RoboDK station: Pick&Place_UR5e.rdk

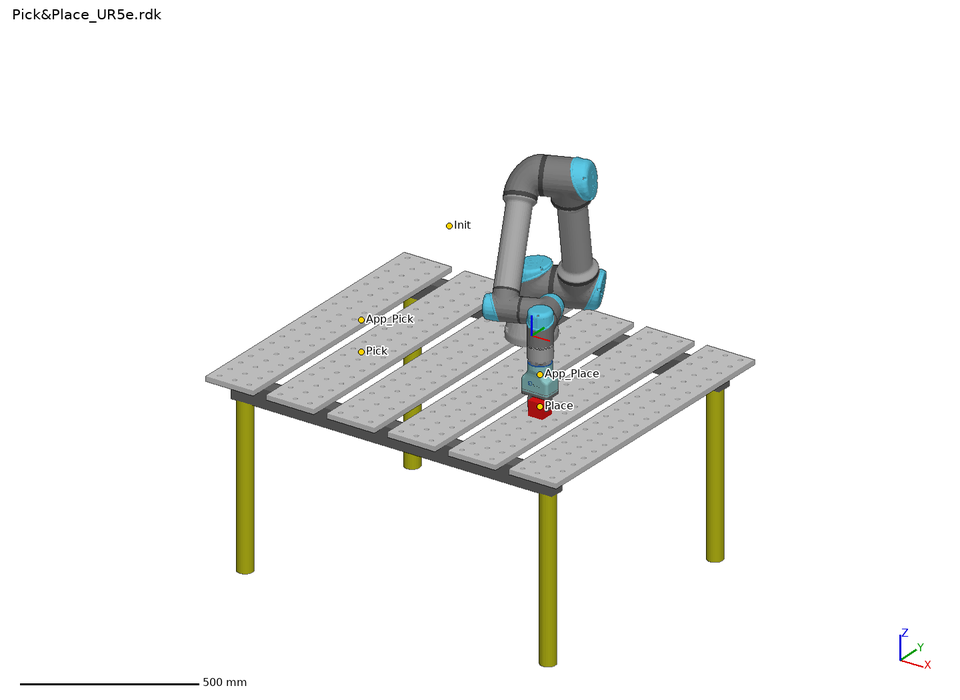
[picture v0: the station drawn from its stored meshes, robots at their saved joint values, targets as dots, program paths as lines]
Station Pick&Place_UR5e (saved by RoboDK 5.9.2). Poses are relative to the parent item; angles as X-Y-Z fixed-axis rotations.
  - frame UR5e Base at (0, 0, 0) mm
    - robot UR5e: 6 axes, payload 5 kg, reach 850 mm, repeatability 0.03 mm, weight 18.4 kg
        modified DH rows (alpha deg, a mm, theta deg, d mm): 0, 0, 0, 162.5; 90, 0, 180, 0; 0, 425, 0, 0; 0, 392.25, 0, 133.3; -90, 0, 0, 99.7; 90, 0, 180, 99.6
        joint limits [-360, -360, -360, -360, -360, -360] to [360, 360, 360, 360, 360, 360]; home [0, -90, -90, 0, 90, 0]; saved at [112.503, -72.13, 120.987, -138.858, -90, 202.503]
      - tool 2FG7, TCP at (0, 0, 147) mm, size 90 x 74.9 x 156.3 mm
  - frame World at (0, 0, 0) mm
    - object Table at (0, 0, 0) mm, size 1193.8 x 965.2 x 609.6 mm, geometry from welding_table.sld
      - object cube at (310, -400, 25) mm, rotated rx 180 ry 0 rz 0 deg, size 48.4 x 48.4 x 48.4 mm, geometry from cube.stl
    - target Init (joint target) at (0, -400, 500) mm, rotated rx 90 ry 0 rz 0 deg; joints [29.661, -137.472, 144.719, -187.246, -29.661, 180] of UR5e
    - target App_Pick (joint target) at (-300, -400, 125) mm, rotated rx 180 ry 0 rz 0 deg; joints [37.668, -82.892, 115.718, -122.826, -90, 127.668] of UR5e
    - target Pick (joint target) at (-300, -400, 25) mm, rotated rx 180 ry 0 rz 0 deg; joints [37.668, -72.781, 121.964, -139.182, -90, 127.668] of UR5e
    - target App_Place (joint target) at (310, -400, 125) mm, rotated rx 180 ry 0 rz 0 deg; joints [112.503, -82.104, 114.797, -122.693, -90, 202.503] of UR5e
    - target Place (joint target) at (310, -400, 25) mm, rotated rx 180 ry 0 rz 0 deg; joints [112.503, -72.13, 120.987, -138.858, -90, 202.503] of UR5e
